Yaskawa INFORM job: INIT_ROS.JBI

/JOB
//NAME INIT_ROS
//POS
///NPOS 0,0,0,0,0,0
//INST
///DATE 2013/07/15 15:32
///ATTR SC,RW
///GROUP1 RB1
NOP
DOUT OT#(890) OFF
DOUT OT#(889) OFF
TIMER T=0.05
SKILLSND "ROS-START"
DOUT OT#(889) ON
WAIT OT#(890)=ON
DOUT OT#(889) OFF
SKILLSND "ROS-STOP"
END
